{attribute 'qualified_only'}
VAR_GLOBAL
	bEnableSwitch : BOOL;
	bModeSwitch : BOOL;
	bStartSwitch : BOOL;

END_VAR

(* stored: Version 1.1.0.1, ProductVersion 3.1.4024.10
   GVL input: Id {8f99161b-15cb-4c9b-a85c-f8e8d6297275} *)
